FUNCTION_BLOCK Plant (* Composite Function Block Type *)
  (* Standard: 61499-2 *)
  (* Version 0.0, 12/12/2023, Cheyan, Schneider Electric, template *)
  PACKAGE Main;
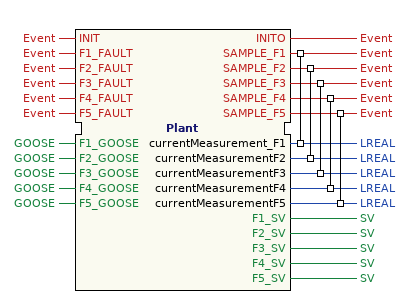
  EVENT_INPUT
    INIT; (* Initialization Request *)
    F1_FAULT;
    F2_FAULT;
    F3_FAULT;
    F4_FAULT;
    F5_FAULT;
  END_EVENT
  EVENT_OUTPUT
    INITO; (* Initialization Confirm *)
    SAMPLE_F1 WITH currentMeasurement_F1;
    SAMPLE_F2 WITH currentMeasurementF2;
    SAMPLE_F3 WITH currentMeasurementF3;
    SAMPLE_F4 WITH currentMeasurementF4;
    SAMPLE_F5 WITH currentMeasurementF5;
  END_EVENT
  VAR_OUTPUT
    currentMeasurement_F1 : LREAL; (* Output event qualifier *)
    currentMeasurementF2 : LREAL; (* Output event qualifier *)
    currentMeasurementF3 : LREAL; (* Output event qualifier *)
    currentMeasurementF4 : LREAL; (* Output event qualifier *)
    currentMeasurementF5 : LREAL; (* Output event qualifier *)
  END_VAR
  SOCKETS
    F1_GOOSE : GOOSE;
    F2_GOOSE : GOOSE;
    F3_GOOSE : GOOSE;
    F4_GOOSE : GOOSE;
    F5_GOOSE : GOOSE;
  END_SOCKETS
  PLUGS
    F1_SV : SV;
    F2_SV : SV;
    F3_SV : SV;
    F4_SV : SV;
    F5_SV : SV;
  END_PLUGS
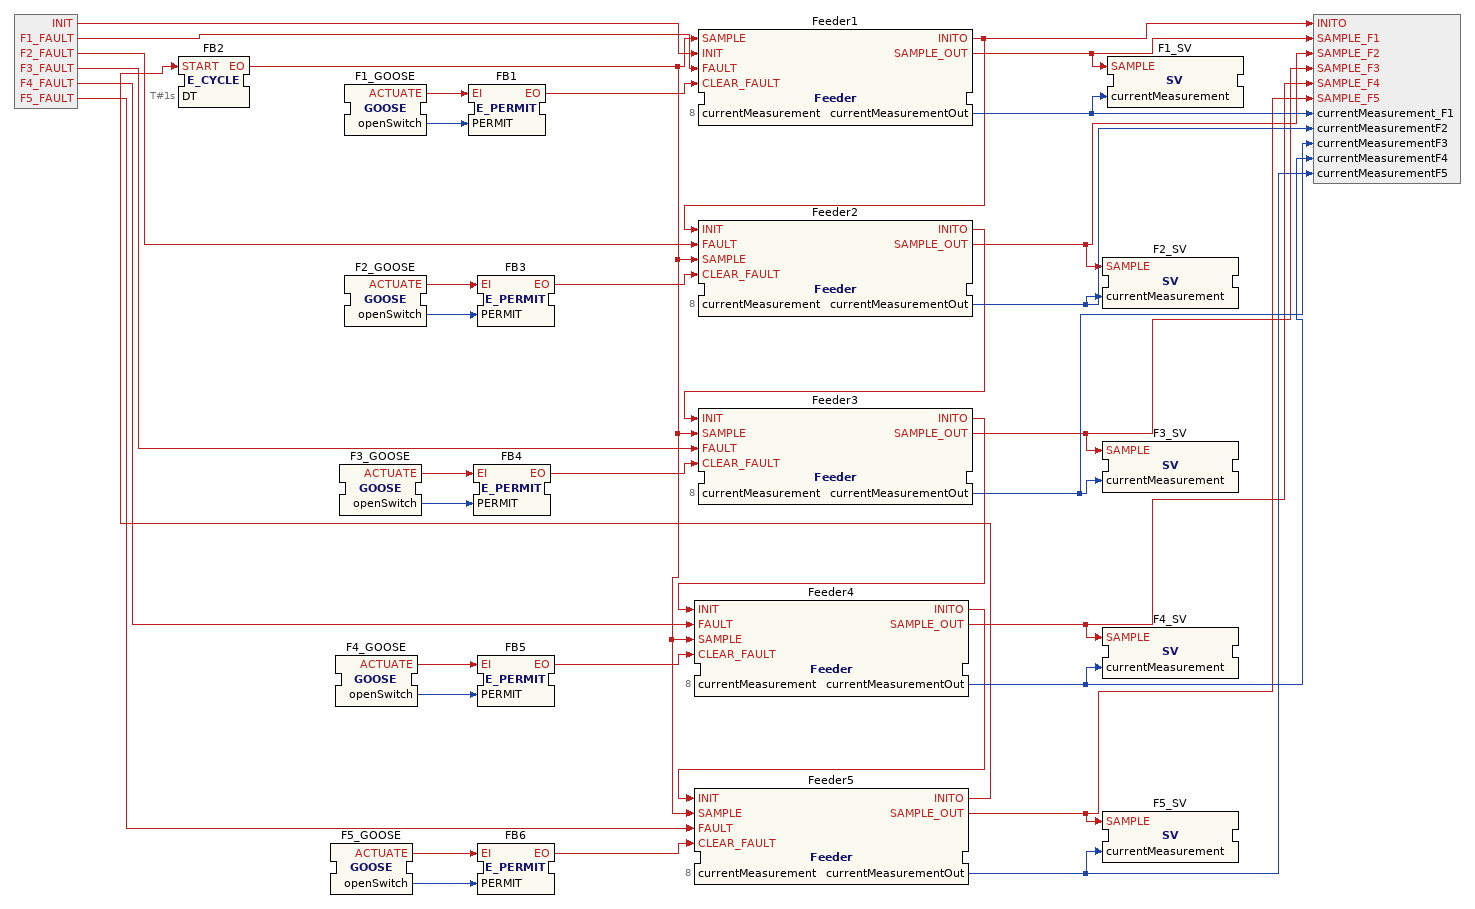
  FBS
    Feeder1 : Feeder(currentMeasurement := 8);
    FB2 : E_CYCLE(DT := T#1s);
    Feeder2 : Feeder(currentMeasurement := 8);
    Feeder3 : Feeder(currentMeasurement := 8);
    Feeder4 : Feeder(currentMeasurement := 8);
    Feeder5 : Feeder(currentMeasurement := 8);
    FB1 : E_PERMIT;
    FB3 : E_PERMIT;
    FB4 : E_PERMIT;
    FB5 : E_PERMIT;
    FB6 : E_PERMIT;
  END_FBS
  EVENT_CONNECTIONS
    FB2.EO TO Feeder1.SAMPLE;
    INIT TO Feeder1.INIT;
    Feeder1.INITO TO Feeder2.INIT;
    Feeder2.INITO TO Feeder3.INIT;
    Feeder3.INITO TO Feeder4.INIT;
    Feeder4.INITO TO Feeder5.INIT;
    Feeder5.INITO TO FB2.START;
    F1_FAULT TO Feeder1.FAULT;
    F2_FAULT TO Feeder2.FAULT;
    FB2.EO TO Feeder2.SAMPLE;
    FB2.EO TO Feeder3.SAMPLE;
    F3_FAULT TO Feeder3.FAULT;
    F4_FAULT TO Feeder4.FAULT;
    FB2.EO TO Feeder4.SAMPLE;
    FB2.EO TO Feeder5.SAMPLE;
    F5_FAULT TO Feeder5.FAULT;
    Feeder1.SAMPLE_OUT TO SAMPLE_F1;
    Feeder1.INITO TO INITO;
    Feeder2.SAMPLE_OUT TO SAMPLE_F2;
    Feeder3.SAMPLE_OUT TO SAMPLE_F3;
    Feeder4.SAMPLE_OUT TO SAMPLE_F4;
    Feeder5.SAMPLE_OUT TO SAMPLE_F5;
    Feeder1.SAMPLE_OUT TO F1_SV.SAMPLE;
    Feeder2.SAMPLE_OUT TO F2_SV.SAMPLE;
    Feeder3.SAMPLE_OUT TO F3_SV.SAMPLE;
    Feeder4.SAMPLE_OUT TO F4_SV.SAMPLE;
    Feeder5.SAMPLE_OUT TO F5_SV.SAMPLE;
    F1_GOOSE.ACTUATE TO FB1.EI;
    FB1.EO TO Feeder1.CLEAR_FAULT;
    F2_GOOSE.ACTUATE TO FB3.EI;
    FB3.EO TO Feeder2.CLEAR_FAULT;
    F3_GOOSE.ACTUATE TO FB4.EI;
    FB4.EO TO Feeder3.CLEAR_FAULT;
    F4_GOOSE.ACTUATE TO FB5.EI;
    FB5.EO TO Feeder4.CLEAR_FAULT;
    F5_GOOSE.ACTUATE TO FB6.EI;
    FB6.EO TO Feeder5.CLEAR_FAULT;
  END_CONNECTIONS
  DATA_CONNECTIONS
    Feeder1.currentMeasurementOut TO currentMeasurement_F1;
    Feeder2.currentMeasurementOut TO currentMeasurementF2;
    Feeder3.currentMeasurementOut TO currentMeasurementF3;
    Feeder4.currentMeasurementOut TO currentMeasurementF4;
    Feeder5.currentMeasurementOut TO currentMeasurementF5;
    Feeder1.currentMeasurementOut TO F1_SV.currentMeasurement;
    Feeder2.currentMeasurementOut TO F2_SV.currentMeasurement;
    Feeder3.currentMeasurementOut TO F3_SV.currentMeasurement;
    Feeder4.currentMeasurementOut TO F4_SV.currentMeasurement;
    Feeder5.currentMeasurementOut TO F5_SV.currentMeasurement;
    F1_GOOSE.openSwitch TO FB1.PERMIT;
    F2_GOOSE.openSwitch TO FB3.PERMIT;
    F3_GOOSE.openSwitch TO FB4.PERMIT;
    F4_GOOSE.openSwitch TO FB5.PERMIT;
    F5_GOOSE.openSwitch TO FB6.PERMIT;
  END_CONNECTIONS
END_FUNCTION_BLOCK
